Yaskawa INFORM job: R1_Z(FRONIUS).JBI

/JOB
//NAME R1_Z(FRONIUS)
///FOLDERNAME INNE
//POS
///NPOS 2,2,0,0,0,0
///TOOL 0
///POSTYPE PULSE
///PULSE
C00000=-92187,-144923,-105356,21900,71569,48314
C00001=-92048,-43024,39511,34235,38461,39008
BC00000=175633,64134,290874
BC00001=175633,64134,864480
//INST
///DATE 2023/10/04 15:16
///ATTR SC,RW
///GROUP1 RB1,BS1
NOP
MOVJ C00000 BC00000 VJ=0.78
MOVJ C00001 BC00001 VJ=0.78
END
